INTERFACE I_MoverSector EXTENDS __SYSTEM.IQueryInterface

PROPERTY P_SectorsConfig : REFERENCE TO ST_SectorsConfig
GET
END_GET
END_PROPERTY

PROPERTY P_SectorsStatus : REFERENCE TO ST_SectorsStatus
GET
END_GET
END_PROPERTY

END_INTERFACE

(* stored: Version 1.1.0.1
   Itf I_MoverSector: Id {bb3c444d-1dfd-435b-9f58-51fe7de2cced}
   Property P_SectorsConfig: Id {6dcaa843-fc31-43e6-a793-9819b587628c}
   Get Get: Id {c6eb122a-2375-444f-afd0-25c33ac13a47}
   Property P_SectorsStatus: Id {f94961d8-fdcd-47ec-b28b-8627807bb068}
   Get Get: Id {f86aa01c-93fa-47ff-acc5-fa5cfdb00094} *)
